// TwinCAT 3 PLC project Demo
// ProgramVersion: 3.1.4023.0
// libraries:
//   Tc2_Standard, * (Beckhoff Automation GmbH)
//   Tc2_System, * (Beckhoff Automation GmbH)
//   Tc3_Module, * (Beckhoff Automation GmbH)
//   VisuSymbols,3.5.10.0,System
// project tree:
//   DUTs/ XeryonDriveError.TcDUT, XeryonDriveSetting.TcDUT, XeryonDriveStatus.TcDUT
//   / GlobalTextList.TcGTLO, PlcTask.TcTTO, Visualization Manager.TcVMO (not stored)
//   GVLs/ GVL.TcGVL
//   POUs/FB/ XeryonDrive.TcPOU
//   POUs/ MAIN.TcPOU, DRIVE_SETTINGS.TcPOU
//   VISUs/ Visualization.TcVIS
// real-time tasks:
//   TASK PlcTask: cycle T#1ms, priority 20, ADS port 350
// I/O:
//   DEVICE Device 1 (EtherCAT), AmsNetId 172.22.11.1.2.1
//     Box 1 (Drive) [Drive]
//     Box 2 (Drive) [Drive] (disabled)
// variable links:
//   Demo/Demo Instance <-> Device 1 (EtherCAT)/Box 1 (Drive)
//     PlcTask Inputs/MAIN.Drive1.iDriveActualPosition <-> Status/Actual position
//     PlcTask Inputs/MAIN.Drive1.iDriveAmplifiersEnabled <-> Status/Amplifiers enabled
//     PlcTask Inputs/MAIN.Drive1.iDriveBusy <-> Status/Execute ack
//     PlcTask Inputs/MAIN.Drive1.iDriveClosedLoop <-> Status/Closed loop
//     PlcTask Inputs/MAIN.Drive1.iDriveEmergencyStop <-> Status/Emergency stop
//     PlcTask Inputs/MAIN.Drive1.iDriveEncoderError <-> Status/Encoder error
//     PlcTask Inputs/MAIN.Drive1.iDriveEncoderIndex <-> Status/Encoder index
//     PlcTask Inputs/MAIN.Drive1.iDriveEncoderValid <-> Status/Encoder valid
//     PlcTask Inputs/MAIN.Drive1.iDriveEndStop <-> Status/End stop
//     PlcTask Inputs/MAIN.Drive1.iDriveErrorCompensation <-> Status/Error compensation
//     PlcTask Inputs/MAIN.Drive1.iDriveErrorLimit <-> Status/Error limit
//     PlcTask Inputs/MAIN.Drive1.iDriveForceZero <-> Status/Force zero
//     PlcTask Inputs/MAIN.Drive1.iDriveLeftEndStop <-> Status/Left end stop
//     PlcTask Inputs/MAIN.Drive1.iDriveMotorOn <-> Status/Motor on
//     PlcTask Inputs/MAIN.Drive1.iDrivePositionFail <-> Status/Position fail
//     PlcTask Inputs/MAIN.Drive1.iDrivePositionReached <-> Status/Position reached
//     PlcTask Inputs/MAIN.Drive1.iDriveRightEndStop <-> Status/Right end stop
//     PlcTask Inputs/MAIN.Drive1.iDriveSafetyTimeoutTriggered <-> Status/Safety timeout
//     PlcTask Inputs/MAIN.Drive1.iDriveScanning <-> Status/Scanning
//     PlcTask Inputs/MAIN.Drive1.iDriveSearchingIndex <-> Status/Searching index
//     PlcTask Inputs/MAIN.Drive1.iDriveSearchingOptimalFrequency <-> Status/Searching optimal frequency
//     PlcTask Inputs/MAIN.Drive1.iDriveSlot <-> Status/Slot
//     PlcTask Inputs/MAIN.Drive1.iDriveThermalProtection1 <-> Status/Thermal protection 1
//     PlcTask Inputs/MAIN.Drive1.iDriveThermalProtection2 <-> Status/Thermal protection 2
//     PlcTask Outputs/MAIN.Drive1.qCommand <-> Position/Command
//     PlcTask Outputs/MAIN.Drive1.qDriveAcc <-> Position/Acceleration
//     PlcTask Outputs/MAIN.Drive1.qDriveDec <-> Position/Deceleration
//     PlcTask Outputs/MAIN.Drive1.qDriveSpeed <-> Position/Speed
//     PlcTask Outputs/MAIN.Drive1.qDriveTargetPos <-> Position/Target position
//     PlcTask Outputs/MAIN.Drive1.qExecute <-> Position/Execute
//   Demo/Demo Instance <-> Device 1 (EtherCAT)/Box 2 (Drive)
//     PlcTask Inputs/MAIN.Drive2.iDriveActualPosition <-> Status/Actual position
//     PlcTask Inputs/MAIN.Drive2.iDriveAmplifiersEnabled <-> Status/Amplifiers enabled
//     PlcTask Inputs/MAIN.Drive2.iDriveBusy <-> Status/Execute ack
//     PlcTask Inputs/MAIN.Drive2.iDriveClosedLoop <-> Status/Closed loop
//     PlcTask Inputs/MAIN.Drive2.iDriveEmergencyStop <-> Status/Emergency stop
//     PlcTask Inputs/MAIN.Drive2.iDriveEncoderError <-> Status/Encoder error
//     PlcTask Inputs/MAIN.Drive2.iDriveEncoderIndex <-> Status/Encoder index
//     PlcTask Inputs/MAIN.Drive2.iDriveEncoderValid <-> Status/Encoder valid
//     PlcTask Inputs/MAIN.Drive2.iDriveEndStop <-> Status/End stop
//     PlcTask Inputs/MAIN.Drive2.iDriveErrorCompensation <-> Status/Error compensation
//     PlcTask Inputs/MAIN.Drive2.iDriveErrorLimit <-> Status/Error limit
//     PlcTask Inputs/MAIN.Drive2.iDriveForceZero <-> Status/Force zero
//     PlcTask Inputs/MAIN.Drive2.iDriveLeftEndStop <-> Status/Left end stop
//     PlcTask Inputs/MAIN.Drive2.iDriveMotorOn <-> Status/Motor on
//     PlcTask Inputs/MAIN.Drive2.iDrivePositionFail <-> Status/Position fail
//     PlcTask Inputs/MAIN.Drive2.iDrivePositionReached <-> Status/Position reached
//     PlcTask Inputs/MAIN.Drive2.iDriveRightEndStop <-> Status/Right end stop
//     PlcTask Inputs/MAIN.Drive2.iDriveSafetyTimeoutTriggered <-> Status/Safety timeout
//     PlcTask Inputs/MAIN.Drive2.iDriveScanning <-> Status/Scanning
//     PlcTask Inputs/MAIN.Drive2.iDriveSearchingIndex <-> Status/Searching index
//     PlcTask Inputs/MAIN.Drive2.iDriveSearchingOptimalFrequency <-> Status/Searching optimal frequency
//     PlcTask Inputs/MAIN.Drive2.iDriveSlot <-> Status/Slot
//     PlcTask Inputs/MAIN.Drive2.iDriveThermalProtection1 <-> Status/Thermal protection 1
//     PlcTask Inputs/MAIN.Drive2.iDriveThermalProtection2 <-> Status/Thermal protection 2
//     PlcTask Outputs/MAIN.Drive2.qCommand <-> Position/Command
//     PlcTask Outputs/MAIN.Drive2.qDriveAcc <-> Position/Acceleration
//     PlcTask Outputs/MAIN.Drive2.qDriveDec <-> Position/Deceleration
//     PlcTask Outputs/MAIN.Drive2.qDriveSpeed <-> Position/Speed
//     PlcTask Outputs/MAIN.Drive2.qDriveTargetPos <-> Position/Target position
//     PlcTask Outputs/MAIN.Drive2.qExecute <-> Position/Execute

CONFIGURATION Demo
    RESOURCE PLC ON TwinCAT3
        TASK PlcTask(INTERVAL := T#1ms, PRIORITY := 20);
        PROGRAM MAIN WITH PlcTask : MAIN;
    END_RESOURCE
END_CONFIGURATION

// ---- DUTs/XeryonDriveError.TcDUT
{attribute 'qualified_only'}
{attribute 'strict'}
{attribute 'to_string'}
TYPE XeryonDriveError :
(
	NO_ERROR := 0,	
	LIMIT_HIT := 1,
	NO_INDEX := 2,
	THERMAL_1 := 3,
	THERMAL_2 := 4,
	ENCODER_ERROR := 5,
	SAFETY_TIMEOUT := 6,
	ERROR_LIMIT := 7,
	ESTOP := 8,
	POS_FAIL := 9,
	DRIVE_DISABLED := 10
);
END_TYPE

// ---- DUTs/XeryonDriveSetting.TcDUT
TYPE XeryonDriveSetting :
STRUCT
	setting : STRING(5);
	value : DINT;
END_STRUCT
END_TYPE

// ---- DUTs/XeryonDriveStatus.TcDUT
{attribute 'qualified_only'}
{attribute 'strict'}
{attribute 'to_string'}
TYPE XeryonDriveStatus :
(	
	Waiting := 0,
	Ready := 1,
	Error := 2,
	SoftError := 3
);
END_TYPE

// ---- GVLs/GVL.TcGVL
{attribute 'qualified_only'}
VAR_GLOBAL	
	Drive1Settings: ARRAY [0..1] OF XeryonDriveSetting;
	Drive2Settings: ARRAY [0..1] OF XeryonDriveSetting;
	Drive3Settings: ARRAY [0..1] OF XeryonDriveSetting;
	Drive4Settings: ARRAY [0..1] OF XeryonDriveSetting;
END_VAR

// ---- POUs/MAIN.TcPOU
PROGRAM MAIN
VAR
	Drive1 : XeryonDrive;
	Drive2 : XeryonDrive;
	Drive3 : XeryonDrive;
	Drive4 : XeryonDrive;
	
	drive1Enable : BOOL;
	drive1EnableOld : BOOL;
	drive1Index : BOOL;
	drive1MoveAbs : BOOL;	
	drive1Dpos : BOOL;		
	drive1Halt : BOOL;
	drive1Stop : BOOL;	
	drive2ResetEncoder : BOOL;	
	drive1ResetEncoder : BOOL;	
	drive1Reset : BOOL;	
	drive1MoveP : BOOL;	
	drive1MoveN : BOOL;		
	drive1JogP : BOOL;	
	drive1JogN : BOOL;	
	drive1Init : BOOL;
	
	drive1State : INT;
	drive1Target : DINT;
	drive1Speed: UDINT := 1000000;
	drive1Acc: UINT := 65535;
	drive1Dec: UINT := 3500;
	drive1ErrorString: STRING;
	
	
	
	drive2Enable : BOOL;
	drive2EnableOld : BOOL;
	drive2Index : BOOL;
	drive2MoveAbs : BOOL;		
	drive2Dpos : BOOL;	
	drive2Halt : BOOL;
	drive2Stop : BOOL;	
	drive2Reset : BOOL;	
	drive2JogP : BOOL;	
	drive2JogN : BOOL;	
	drive2Init : BOOL;
	
	drive2State : INT;
	drive2Target : DINT;
	drive2Speed: UDINT := 150000;
	drive2Acc: UINT := 10000;
	drive2Dec: UINT := 10000;
	
	
	drive3Enable : BOOL;
	drive3EnableOld : BOOL;
	drive3Index : BOOL;
	drive3MoveAbs : BOOL;		
	drive3Dpos : BOOL;		
	drive3Halt : BOOL;
	drive3Stop : BOOL;	
	drive3Reset : BOOL;	
	drive3JogP : BOOL;	
	drive3JogN : BOOL;	
	drive3Init : BOOL;
	
	drive3State : INT;
	drive3Target : DINT;
	drive3Speed: UDINT := 150000;
	drive3Acc: UINT := 10000;
	drive3Dec: UINT := 10000;


	drive4Enable : BOOL;
	drive4EnableOld : BOOL;
	drive4Index : BOOL;
	drive4MoveAbs : BOOL;		
	drive4Dpos : BOOL;		
	drive4Halt : BOOL;
	drive4Stop : BOOL;	
	drive4Reset : BOOL;	
	drive4JogP : BOOL;	
	drive4JogN : BOOL;	
	drive4Init : BOOL;
	
	drive4State : INT;
	drive4Target : DINT;
	drive4Speed: UDINT := 150000;
	drive4Acc: UINT := 10000;
	drive4Dec: UINT := 10000;

	
	target_min : DINT;
	target_max : DINT;
	
	speed_min : DINT;
	speed_max : DINT;
	
	acc_min : DINT;
	acc_max : DINT;
	dec_min : DINT;
	dec_max : DINT;
	
	drive2ErrorString: STRING;
	drive3ErrorString: STRING;
	drive4ErrorString: STRING;
	dpos: DINT;
	drive2MoveN: BOOL;
	Halt: INT;
	drive2MoveP: BOOL;
END_VAR

DRIVE_SETTINGS();

Drive1();
Drive2();
Drive3();
Drive4();
drive1ErrorString := TO_STRING(Drive1.Error);
drive2ErrorString := TO_STRING(Drive2.Error);
drive3ErrorString := TO_STRING(Drive3.Error);
drive4ErrorString := TO_STRING(Drive4.Error);
// DEMO Drive 1
CASE drive1State OF
	0:
		IF(drive1JogP) THEN
			drive1State := 10;
		END_IF
		IF(drive1JogN) THEN
			drive1State := 14;
		END_IF
		IF(drive1MoveP) THEN
			drive1State := 17;
		END_IF
		IF(drive1MoveN) THEN
			drive1State := 20;
		END_IF
		IF(drive1Init) THEN
			drive1State := 9;
		END_IF
		IF(drive1MoveAbs) THEN
			drive1State := 2;
		END_IF
		IF(drive1Index) THEN
			drive1State := 1;
		END_IF
		IF(drive1Dpos) THEN
			drive1State := 8;
		END_IF
	1:
		IF(NOT drive1Index) THEN
			IF(Drive1.Index(drive1Target > 0, drive1Speed, drive1Acc, drive1Dec)<> XeryonDriveStatus.Waiting) THEN
				drive1State := 0;
			END_IF
		END_IF
	2:
		IF(Drive1.MoveAbsolute(dpos, drive1Speed, drive1Acc, drive1Dec)<> XeryonDriveStatus.Waiting) THEN
			IF(dpos < 921600) THEN
				dpos:=dpos+25600;
			ELSE
				dpos := 1000;
			END_IF
			drive1State := 0;
		END_IF
	3:
		IF(Drive1.MoveAbsolute(-40000, drive1Speed, drive1Acc, drive1Dec)<> XeryonDriveStatus.Waiting) THEN
			drive1State := 4;
		END_IF
	4: 
		IF(Drive1.MoveAbsolute(0, drive1Speed, drive1Acc, drive1Dec)<> XeryonDriveStatus.Waiting) THEN
			drive1State := 5;
		END_IF
	5: 
		IF(Drive1.MoveAbsolute(-10000, drive1Speed, drive1Acc, drive1Dec)<> XeryonDriveStatus.Waiting) THEN
			drive1State := 6;
		END_IF
	6: 
		IF(Drive1.MoveAbsolute(0, drive1Speed, drive1Acc, drive1Dec)<> XeryonDriveStatus.Waiting) THEN
			drive1State := 7;
		END_IF		
	7: 
		IF(Drive1.MoveAbsolute(-5000, drive1Speed, drive1Acc, drive1Dec)<> XeryonDriveStatus.Waiting) THEN
			drive1State := 0;
		END_IF
	8:
		IF(NOT drive1Dpos) THEN
			IF(Drive1.MoveAbsolute(drive1Target, drive1Speed, drive1Acc, drive1Dec)<> XeryonDriveStatus.Waiting) THEN
				drive1State := 0;
			END_IF
		END_IF
	9:
		IF(Drive1.Init(GVL.Drive1Settings) = TRUE) THEN
			drive1State := 0;
		END_IF
	10:
		IF(Drive1.Scan(TRUE, drive1Speed, drive1Acc, drive1Dec) <>  XeryonDriveStatus.Waiting) THEN
			drive1State := 12;
		END_IF
	12: //TBD GST : why is this state needed???
		IF(NOT drive1JogP) THEN
			drive1State := 13;
		END_IF
	13:
		IF(Drive1.Halt() <>  XeryonDriveStatus.Waiting) THEN
			drive1State := 0;
		END_IF
	14:
		IF(Drive1.Scan(FALSE, drive1Speed, drive1Acc, drive1Dec) <>  XeryonDriveStatus.Waiting) THEN
			drive1State := 15;
		END_IF
	15:
		IF(NOT drive1JogN) THEN
			drive1State := 16;
		END_IF
	16:
		IF(Drive1.Halt() <>  XeryonDriveStatus.Waiting) THEN
			drive1State := 0;
		END_IF
		
	17:
		IF(Drive1.MoveOpen(TRUE) <>  XeryonDriveStatus.Waiting) THEN
			drive1State := 18;
		END_IF
	18:
		IF(NOT drive1MoveP) THEN
			drive1State := 19;
		END_IF
	19:
		IF(Drive1.Halt() <>  XeryonDriveStatus.Waiting) THEN
			drive1State := 0;
		END_IF
	20:
		IF(Drive1.MoveOpen(FALSE) <>  XeryonDriveStatus.Waiting) THEN
			drive1State := 21;
		END_IF
	21:
		IF(NOT drive1MoveN) THEN
			drive1State := 22;
		END_IF
	22:
		IF(Drive1.Halt() <>  XeryonDriveStatus.Waiting) THEN
			drive1State := 0;
		END_IF	
			
END_CASE

IF(drive1Halt) THEN
	Drive1.Halt();
END_IF
IF(drive1Enable <> drive1EnableOld) THEN	
	IF(Drive1.Enable(drive1Enable) <> XeryonDriveStatus.Waiting) THEN
		drive1EnableOld := drive1Enable;	
	END_IF
END_IF
IF(drive1Stop) THEN
	Drive1.Stop();
END_IF
IF(drive1Reset) THEN
	Drive1.Reset();
END_IF
IF(drive1ResetEncoder) THEN
	Drive1.ResetEncoder();
END_IF

// DEMO Drive 2
CASE drive2State OF
	0:
		IF(drive2JogP) THEN
			drive2State := 10;
		END_IF
		IF(drive2JogN) THEN
			drive2State := 14;
		END_IF
		IF(drive2MoveP) THEN
			drive2State := 17;
		END_IF
		IF(drive2MoveN) THEN
			drive2State := 20;
		END_IF
		IF(drive2Init) THEN
			drive2State := 9;
		END_IF
		IF(drive2MoveAbs) THEN
			drive2State := 2;
		END_IF
		IF(drive2Index) THEN
			drive2State := 1;
		END_IF
		IF(drive2Dpos) THEN
			drive2State := 8;
		END_IF
	1:
		IF(NOT drive2Index) THEN
			IF(Drive2.Index(drive2Target > 0, drive2Speed, drive2Acc, drive2Dec)<> XeryonDriveStatus.Waiting) THEN
				drive2State := 0;
			END_IF
		END_IF
	2:
		IF(Drive2.MoveAbsolute(40000, drive2Speed, drive2Acc, drive2Dec)<> XeryonDriveStatus.Waiting) THEN
			drive2State := 3;
		END_IF
	3: 
		IF(Drive2.MoveAbsolute(0, drive2Speed, drive2Acc, drive2Dec)<> XeryonDriveStatus.Waiting) THEN
			drive2State := 4;
		END_IF
	4: 
		IF(Drive2.MoveAbsolute(-40000, drive2Speed, drive2Acc, drive2Dec)<> XeryonDriveStatus.Waiting) THEN
			drive2State := 5;
		END_IF
	5: 
		IF(Drive2.MoveAbsolute(-10000, drive2Speed, drive2Acc, drive2Dec)<> XeryonDriveStatus.Waiting) THEN
			drive2State := 6;
		END_IF
	6: 
		IF(Drive2.MoveAbsolute(-5000, drive2Speed, drive2Acc, drive2Dec)<> XeryonDriveStatus.Waiting) THEN
			drive2State := 7;
		END_IF		
	7: 
		IF(Drive2.MoveAbsolute(0, drive2Speed, drive2Acc, drive2Dec)<> XeryonDriveStatus.Waiting) THEN
			drive2State := 0;
		END_IF
	8:
		IF(NOT drive2Dpos) THEN
			IF(Drive2.MoveAbsolute(drive2Target, drive2Speed, drive2Acc, drive2Dec)<> XeryonDriveStatus.Waiting) THEN
				drive2State := 0;
			END_IF
		END_IF
	9:
		IF(Drive2.Init(GVL.Drive2Settings) = TRUE) THEN
			drive2State := 0;
		END_IF
	10:
		IF(Drive2.Scan(TRUE, drive2Speed, drive2Acc, drive2Dec) <>  XeryonDriveStatus.Waiting) THEN
			drive2State := 12;
		END_IF
	12:
		IF(NOT drive2JogP) THEN
			drive2State := 13;
		END_IF
	13:
		IF(Drive2.Halt() <>  XeryonDriveStatus.Waiting) THEN
			drive2State := 0;
		END_IF
	14:
		IF(Drive2.Scan(FALSE, drive2Speed, drive2Acc, drive2Dec) <>  XeryonDriveStatus.Waiting) THEN
			drive2State := 15;
		END_IF
	15:
		IF(NOT drive2JogN) THEN
			drive2State := 16;
		END_IF
	16:
		IF(Drive2.Halt() <>  XeryonDriveStatus.Waiting) THEN
			drive2State := 0;
		END_IF
	17:
		IF(Drive2.MoveOpen(TRUE) <>  XeryonDriveStatus.Waiting) THEN
			drive2State := 18;
		END_IF
	18:
		IF(NOT drive2MoveP) THEN
			drive2State := 19;
		END_IF
	19:
		IF(Drive2.Halt() <>  XeryonDriveStatus.Waiting) THEN
			drive2State := 0;
		END_IF
	20:
		IF(Drive2.MoveOpen(FALSE) <>  XeryonDriveStatus.Waiting) THEN
			drive2State := 21;
		END_IF
	21:
		IF(NOT drive2MoveN) THEN
			drive2State := 22;
		END_IF
	22:
		IF(Drive2.Halt() <>  XeryonDriveStatus.Waiting) THEN
			drive2State := 0;
		END_IF
END_CASE

IF(drive2Halt) THEN
	Drive2.Halt();
END_IF
IF(drive2Enable <> drive2EnableOld) THEN
	IF(Drive2.Enable(drive2Enable) <> XeryonDriveStatus.Waiting) THEN
		drive2EnableOld := drive2Enable;	
	END_IF
END_IF
IF(drive2Stop) THEN
	Drive2.Stop();
END_IF
IF(drive2Reset) THEN
	Drive2.Reset();
END_IF
IF(drive2ResetEncoder) THEN
	Drive2.ResetEncoder();
END_IF

// DEMO Drive 3
CASE drive3State OF
	0:
		IF(drive3JogP) THEN
			drive3State := 10;
		END_IF
		IF(drive3JogN) THEN
			drive3State := 14;
		END_IF
		IF(drive3Init) THEN
			drive3State := 9;
		END_IF
		IF(drive3MoveAbs) THEN
			drive3State := 2;
		END_IF
		IF(drive3Index) THEN
			drive3State := 1;
		END_IF
		IF(drive3Dpos) THEN
			drive3State := 8;
		END_IF
	1:
		IF(NOT drive3Index) THEN
			IF(Drive3.Index(drive3Target  > 0, drive3Speed, drive3Acc, drive3Dec) <> XeryonDriveStatus.Waiting) THEN
				drive3State := 0;
			END_IF
		END_IF
	2:
		IF(Drive3.MoveAbsolute(40000, drive3Speed, drive3Acc, drive3Dec) <> XeryonDriveStatus.Waiting) THEN
			drive3State := 3;
		END_IF
	3: 
		IF(Drive3.MoveAbsolute(0, drive3Speed, drive3Acc, drive3Dec) <> XeryonDriveStatus.Waiting) THEN
			drive3State := 4;
		END_IF
	4: 
		IF(Drive3.MoveAbsolute(-40000, drive3Speed, drive3Acc, drive3Dec) <> XeryonDriveStatus.Waiting) THEN
			drive3State := 5;
		END_IF
	5: 
		IF(Drive3.MoveAbsolute(15000, drive3Speed, drive3Acc, drive3Dec) <> XeryonDriveStatus.Waiting) THEN
			drive3State := 6;
		END_IF
	6: 
		IF(Drive3.MoveAbsolute(-15000, drive3Speed, drive3Acc, drive3Dec) <> XeryonDriveStatus.Waiting) THEN
			drive3State := 7;
		END_IF		
	7: 
		IF(Drive3.MoveAbsolute(0, drive3Speed, drive3Acc, drive3Dec) <> XeryonDriveStatus.Waiting) THEN
			drive3State := 0;
		END_IF
	8:
		IF(NOT drive3Dpos) THEN
			IF(Drive3.MoveAbsolute(drive3Target, drive3Speed, drive3Acc, drive3Dec) <> XeryonDriveStatus.Waiting) THEN
				drive3State := 0;
			END_IF
		END_IF
	9:
		IF(Drive3.Init(GVL.Drive3Settings) = TRUE) THEN
			drive3State := 0;
		END_IF
	10:
		IF(Drive3.Scan(TRUE, drive3Speed, drive3Acc, drive3Dec) <>  XeryonDriveStatus.Waiting) THEN
			drive3State := 12;
		END_IF
	12:
		IF(NOT drive3JogP) THEN
			drive3State := 13;
		END_IF
	13:
		IF(Drive3.Halt() <>  XeryonDriveStatus.Waiting) THEN
			drive3State := 0;
		END_IF
	14:
		IF(Drive3.Scan(FALSE, drive3Speed, drive3Acc, drive3Dec) <>  XeryonDriveStatus.Waiting) THEN
			drive3State := 15;
		END_IF
	15:
		IF(NOT drive3JogN) THEN
			drive3State := 16;
		END_IF
	16:
		IF(Drive3.Halt() <>  XeryonDriveStatus.Waiting) THEN
			drive3State := 0;
		END_IF		
		
END_CASE

IF(drive3Halt) THEN
	Drive3.Halt();
END_IF
IF(drive3Stop) THEN
	Drive3.Stop();
END_IF
IF(drive3Enable <> drive3EnableOld) THEN
	IF(Drive3.Enable(drive3Enable) <> XeryonDriveStatus.Waiting) THEN
		drive3EnableOld := drive3Enable;	
	END_IF
END_IF
IF(drive3Reset) THEN
	Drive3.Reset();
END_IF




// DEMO Drive 4
CASE drive4State OF
	0:
		IF(drive4JogP) THEN
			drive4State := 10;
		END_IF
		IF(drive4JogN) THEN
			drive4State := 14;
		END_IF
		IF(drive4Init) THEN
			drive4State := 9;
		END_IF
		IF(drive4MoveAbs) THEN
			drive4State := 2;
		END_IF
		IF(drive4Index) THEN
			drive4State := 1;
		END_IF
		IF(drive4Dpos) THEN
			drive4State := 8;
		END_IF
	1:
		IF(NOT drive4Index) THEN
			IF(Drive4.Index(drive4Target  > 0, drive4Speed, drive4Acc, drive4Dec) <> XeryonDriveStatus.Waiting) THEN
				drive4State := 0;
			END_IF
		END_IF
	2:
		IF(Drive4.MoveAbsolute(0, drive4Speed, drive4Acc, drive4Dec) <> XeryonDriveStatus.Waiting) THEN
			drive4State := 3;
		END_IF
	3: 
		IF(Drive4.MoveAbsolute(35000, drive4Speed, drive4Acc, drive4Dec) <> XeryonDriveStatus.Waiting) THEN
			drive4State := 4;
		END_IF
	4: 
		IF(Drive4.MoveAbsolute(0, drive4Speed, drive4Acc, drive4Dec) <> XeryonDriveStatus.Waiting) THEN
			drive4State := 5;
		END_IF
	5: 
		IF(Drive4.MoveAbsolute(-35000, drive4Speed, drive4Acc, drive4Dec) <> XeryonDriveStatus.Waiting) THEN
			drive4State := 6;
		END_IF
	6: 
		IF(Drive4.MoveAbsolute(0, drive4Speed, drive4Acc, drive4Dec) <> XeryonDriveStatus.Waiting) THEN
			drive4State := 7;
		END_IF		
	7: 
		IF(Drive4.MoveAbsolute(35000, drive4Speed, drive4Acc, drive4Dec) <> XeryonDriveStatus.Waiting) THEN
			drive4State := 0;
		END_IF
	8:
		IF(NOT drive4Dpos) THEN
			IF(Drive4.MoveAbsolute(drive4Target, drive4Speed, drive4Acc, drive4Dec) <> XeryonDriveStatus.Waiting) THEN
				drive4State := 0;
			END_IF
		END_IF
	9:
		IF(Drive4.Init(GVL.Drive4Settings) = TRUE) THEN
			drive4State := 0;
		END_IF
	10:
		IF(Drive4.Scan(TRUE, drive4Speed, drive4Acc, drive4Dec) <>  XeryonDriveStatus.Waiting) THEN
			drive4State := 12;
		END_IF
	12:
		IF(NOT drive4JogP) THEN
			drive4State := 13;
		END_IF
	13:
		IF(Drive4.Halt() <>  XeryonDriveStatus.Waiting) THEN
			drive4State := 0;
		END_IF
	14:
		IF(Drive4.Scan(FALSE, drive4Speed, drive4Acc, drive4Dec) <>  XeryonDriveStatus.Waiting) THEN
			drive4State := 15;
		END_IF
	15:
		IF(NOT drive4JogN) THEN
			drive4State := 16;
		END_IF
	16:
		IF(Drive4.Halt() <>  XeryonDriveStatus.Waiting) THEN
			drive4State := 0;
		END_IF		
		
END_CASE

IF(drive4Halt) THEN
	Drive4.Halt();
END_IF
IF(drive4Stop) THEN
	Drive4.Stop();
END_IF
IF(drive4Enable <> drive4EnableOld) THEN
	IF(Drive4.Enable(drive4Enable) <> XeryonDriveStatus.Waiting) THEN
		drive4EnableOld := drive4Enable;	
	END_IF
END_IF
IF(drive4Reset) THEN
	Drive4.Reset();
END_IF


target_max := 1843200;
target_min := -1843200;

speed_min := 0;
speed_max := 1000000;


acc_min := 0;
acc_max := 65535;

dec_min := 0;
dec_max := 65535;

END_PROGRAM

// ---- POUs/FB/XeryonDrive.TcPOU
FUNCTION_BLOCK XeryonDrive
VAR_INPUT
END_VAR
VAR_OUTPUT
	ActPosition : DINT;
	Done : BOOL;
	Busy : BOOL;
	HasError : BOOL;
	HasIndex : BOOL;
	Error : XeryonDriveError;
	MotorOn : BOOL;
	LeftEndstop : BOOL;
	RightEndstop : BOOL;
END_VAR
VAR
	iDriveActualPosition AT %I* : DINT;
	iDriveAmplifiersEnabled AT %I* : BOOL;
	iDriveEndStop AT %I* : BOOL;
	iDriveThermalProtection1 AT %I* : BOOL;
	iDriveThermalProtection2 AT %I* : BOOL;
	iDriveForceZero AT %I* : BOOL;
	iDriveMotorOn AT %I* : BOOL;
	iDriveClosedLoop AT %I* : BOOL;
	iDriveEncoderIndex AT %I* : BOOL;
	iDriveEncoderValid AT %I* : BOOL;
	iDriveSearchingIndex AT %I* : BOOL;
	iDrivePositionReached AT %I* : BOOL;
	iDriveErrorCompensation AT %I* : BOOL;
	iDriveEncoderError AT %I* : BOOL;
	iDriveScanning AT %I* : BOOL;
	iDriveLeftEndStop AT %I* : BOOL;
	iDriveRightEndStop AT %I* : BOOL;
	iDriveErrorLimit AT %I* : BOOL;
	iDriveSearchingOptimalFrequency AT %I* : BOOL;
	iDriveSafetyTimeoutTriggered AT %I* : BOOL;
	iDriveBusy AT %I* : BOOL;
	iDriveEmergencyStop AT %I* : BOOL;
	iDrivePositionFail AT %I* : BOOL;
	iDriveSlot AT %I* : USINT;
	
	qDriveTargetPos AT %Q* : DINT;
	qDriveSpeed AT %Q* : DINT;
	qDriveAcc AT %Q* : INT;
	qDriveDec AT %Q* : INT;
	qCommand AT %Q* : STRING(4);
	qExecute AT %Q* : USINT;
	
	
	new_TargetPos : DINT;
	new_Speed : UDINT;
	new_Acc : INT;
	new_Dec : INT;
	new_command : STRING(4);
	
	state : INT := 0;
	command_start : BOOL;
	command_done : BOOL;
	command_irq : BOOL;
	init_state : INT := -1;
	
	has_index : BOOL;
	
END_VAR

has_index := iDriveEncoderValid;
ActPosition := iDriveActualPosition;
MotorOn := iDriveMotorOn;
LeftEndstop := iDriveLeftEndStop;
RightEndstop := iDriveRightEndStop;
HasIndex := has_index;

// Check error bits
IF(iDriveThermalProtection1) THEN
	HasError := TRUE;
	Error := XeryonDriveError.THERMAL_1;
END_IF
IF(iDriveThermalProtection1) THEN
	HasError := TRUE;
	Error := XeryonDriveError.THERMAL_2;
END_IF
IF(iDriveEncoderError) THEN
	HasError := TRUE;
	Error := XeryonDriveError.ENCODER_ERROR;
END_IF
IF(iDriveEmergencyStop) THEN
	HasError := TRUE;
	Error := XeryonDriveError.ESTOP;
END_IF
IF(iDriveErrorLimit) THEN
	HasError := TRUE;
	Error := XeryonDriveError.ERROR_LIMIT;
END_IF

CASE state OF
	0: // Idle
	 	IF(command_irq = TRUE) THEN
			state := 4;
		END_IF
	 	IF(command_start = TRUE) THEN
			state := 1;
		END_IF
		Busy := FALSE;
	1:
		Busy := TRUE;
		Done := FALSE;
		qCommand := new_command;
		qDriveTargetPos := new_TargetPos;
		qDriveSpeed := UDINT_TO_DINT(new_Speed);
		qDriveAcc := new_Acc;
		qDriveDec := new_Dec;
		qExecute := 255;
		command_start := FALSE;
		command_done := FALSE;
		IF(iDriveBusy = TRUE) THEN
			qExecute := 0;
			state := 2;	
		END_IF		
	2:	
		IF(iDriveBusy = FALSE) THEN
			state := 3;	
		END_IF	
	3: 	IF(command_done = TRUE) THEN
			state := 0;			
			Done := TRUE;
		END_IF
	 	IF(command_irq = TRUE) THEN
			state := 4;
		END_IF
	// Interrupt commands 
	4:	
		command_irq := FALSE;
		Busy := TRUE;
		Done := FALSE;
		qCommand := new_command;
		qDriveTargetPos := new_TargetPos;
		qDriveSpeed := UDINT_TO_DINT(new_Speed);
		qDriveAcc := new_Acc;
		qDriveDec := new_Dec;
		qExecute := 255;
		command_start := FALSE;
		command_done := FALSE;
		IF(iDriveBusy = TRUE) THEN
			qExecute := 0;
			state := 5;	
		END_IF		
	5:	IF(iDriveBusy = FALSE) THEN
			qExecute := 0;
			state := 6;	
		END_IF	
	6:
		state := 0;			
		Done := TRUE;
	
END_CASE

METHOD CheckError : BOOL
VAR_INPUT
END_VAR
CheckError := FALSE;
// Only check these two  bits when moving
IF(iDrivePositionFail) THEN
	HasError := TRUE;
	Error := XeryonDriveError.POS_FAIL;
END_IF
IF(iDriveSafetyTimeoutTriggered) THEN
	HasError := TRUE;
	Error := XeryonDriveError.SAFETY_TIMEOUT;
END_IF
IF(HasError) THEN
	CheckError := TRUE;	
END_IF
END_METHOD

ACTION ClearError:
HasError := FALSE;
Error := XeryonDriveError.NO_ERROR;

// Reset the index when clearing the error
IF(iDriveEncoderValid) THEN
	has_index := TRUE;
ELSE
	has_index := FALSE;
END_IF
END_ACTION

METHOD Enable : XeryonDriveStatus
VAR_INPUT
	val : BOOL;
END_VAR
Enable := XeryonDriveStatus.Waiting;
IF(state = 0) OR (state = 3) THEN
	new_command := 'ENBL';
	IF(val) THEN
		new_TargetPos := 1;
	ELSE
		new_TargetPos := 0;
	END_IF
	command_start := TRUE;
	command_irq := TRUE;
END_IF
IF(state = 6) THEN
	command_done := TRUE;
	Enable := XeryonDriveStatus.Ready;
	// Clear error
	IF(val) THEN
		ClearError();
	END_IF	
END_IF
END_METHOD

METHOD Halt : XeryonDriveStatus
VAR_INPUT
END_VAR
Halt := XeryonDriveStatus.Waiting;
IF(state = 0) OR (state = 3)THEN
	new_command := 'HALT';
	command_start := TRUE;
	command_irq := TRUE;
END_IF
IF(state = 6) THEN
	command_done := TRUE;
	Halt := XeryonDriveStatus.Ready;
END_IF
END_METHOD

METHOD Index : XeryonDriveStatus
VAR_INPUT
	Direction : BOOL;
	Velocity : UDINT;
	Acceleration: UINT;
	Deceleration: UINT;
END_VAR
Index := XeryonDriveStatus.Waiting;
IF(state = 0) THEN
	// Only execute when we don't have an active error
	IF(NOT HasError) THEN
		IF(iDriveAmplifiersEnabled) THEN
			new_command := 'INDX';
			IF(Direction) THEN
				new_TargetPos := +1;	
			ELSE
				new_TargetPos := -1;
			END_IF		
			new_Speed := Velocity;
			new_Acc := UINT_TO_INT(Acceleration);
			new_Dec := UINT_TO_INT(Deceleration);
			command_start := TRUE;
		ELSE
			
			HasError := TRUE;
			IF(NOT iDriveAmplifiersEnabled) THEN
				Error := XeryonDriveError.DRIVE_DISABLED;	
			END_IF		
			Index := XeryonDriveStatus.Error;	
		END_IF
	ELSE
		Index := XeryonDriveStatus.Error;
	END_IF
END_IF
IF(state = 3) THEN
	// Normal flow, when index is found --> ready 
	IF(iDriveEncoderValid) THEN
		command_done := TRUE;
		Index := XeryonDriveStatus.Ready;
	END_IF
	
	// When hitting the endstop signal a SoftError, doesn't need a reset, but limit the motion
	IF(iDriveEndstop) THEN
		command_done := TRUE;
		Index := XeryonDriveStatus.SoftError;		
	END_IF
	
	// Handle drive errors
	IF(CheckError()) THEN
		command_done := TRUE;
		Index := XeryonDriveStatus.Error;
	END_IF
END_IF
IF(state = 6) THEN
	Index := XeryonDriveStatus.Ready;
END_IF
END_METHOD

METHOD Init : BOOL
VAR_IN_OUT
	settings : ARRAY[*] OF XeryonDriveSetting;
END_VAR
Init := FALSE;

// Start
IF(init_state = -1) THEN
	init_state := DINT_TO_INT(LOWER_BOUND(settings, 1));
END_IF

IF(init_state >=  LOWER_BOUND(settings, 1)) AND (init_state < UPPER_BOUND(settings, 1))  THEN
	IF(Write(settings[init_state].setting, settings[init_state].value) <> XeryonDriveStatus.Waiting) THEN
		init_state := init_state + 1;
		IF(init_state = UPPER_BOUND(settings, 1)) THEN
			init_state := -1;
			Init := TRUE;
		END_IF
	END_IF
END_IF
END_METHOD

METHOD MoveAbsolute : XeryonDriveStatus
VAR_INPUT
	Position : DINT;
	Velocity : UDINT;
	Acceleration: UINT;
	Deceleration: UINT;
	
END_VAR
MoveAbsolute := XeryonDriveStatus.Waiting;
IF(state = 0) THEN
	// Only execute when we don't have an active error
	IF(NOT HasError) THEN		
		// Check if we have an index
		IF(has_index) AND iDriveAmplifiersEnabled THEN
			new_command := 'DPOS';
			new_TargetPos := Position;
			new_Speed := Velocity;
			new_Acc := UINT_TO_INT(Acceleration);
			new_Dec := UINT_TO_INT(Deceleration);
			command_start := TRUE;
		ELSE
			HasError := TRUE;
			IF(NOT has_index) THEN
				Error := XeryonDriveError.NO_INDEX;	
			END_IF
			IF(NOT iDriveAmplifiersEnabled) THEN
				Error := XeryonDriveError.DRIVE_DISABLED;	
			END_IF

			MoveAbsolute := XeryonDriveStatus.Error;
		END_IF
	ELSE
		MoveAbsolute := XeryonDriveStatus.Error;
	END_IF	
	
END_IF
IF(state = 3) THEN
	
	// Normal flow, when position is reached  --> ready 
	IF(iDrivePositionReached) THEN
		command_done := TRUE;
		MoveAbsolute := XeryonDriveStatus.Ready;
	END_IF
	
	// When hitting the endstop signal a SoftError, doesn't need a reset, but limit the motion
	IF(iDriveEndstop) THEN
		command_done := TRUE;
		MoveAbsolute := XeryonDriveStatus.SoftError;		
	END_IF
	
	// Handle drive errors
	IF(CheckError()) THEN
		command_done := TRUE;
		MoveAbsolute := XeryonDriveStatus.Error;
	END_IF
	
END_IF
IF(state = 6) THEN
	MoveAbsolute := XeryonDriveStatus.Ready;
END_IF
END_METHOD

METHOD MoveOpen : XeryonDriveStatus
VAR_INPUT
	Direction: BOOL;	
END_VAR
MoveOpen := XeryonDriveStatus.Waiting;
IF(state = 0) THEN
	IF( NOT HasError) THEN
		IF iDriveAmplifiersEnabled THEN
			new_command := 'MOVE';
			IF(Direction) THEN
				new_TargetPos := +1;	
			ELSE
				new_TargetPos := -1;
			END_IF
			new_Speed := 0;
			new_Acc := UINT_TO_INT(0);
			new_Dec := UINT_TO_INT(0);
			command_start := TRUE;
		ELSE
			HasError := TRUE;
			IF(NOT iDriveAmplifiersEnabled) THEN
				Error := XeryonDriveError.DRIVE_DISABLED;	
			END_IF		
			MoveOpen := XeryonDriveStatus.Error;	
		END_IF
	ELSE
		MoveOpen := XeryonDriveStatus.Error;
	END_IF	
END_IF
IF(state = 3) THEN
	command_done := TRUE;
	MoveOpen := XeryonDriveStatus.Ready;
END_IF
IF(state = 6) THEN
	MoveOpen := XeryonDriveStatus.Ready;
END_IF
END_METHOD

METHOD Reset : XeryonDriveStatus
VAR_INPUT
END_VAR
Reset := XeryonDriveStatus.Waiting;
IF(state = 0) OR (state = 3) THEN
	new_command := 'RSET';
	command_start := TRUE;
	command_irq := TRUE;
END_IF
IF(state = 6) THEN
	command_done := TRUE;
	Reset := XeryonDriveStatus.Ready;
	
	// Clear errors
	ClearError();
	
	// Clear Index
	has_index := FALSE;
	
END_IF
END_METHOD

METHOD ResetEncoder : XeryonDriveStatus
ResetEncoder := XeryonDriveStatus.Waiting;
IF(state = 0) OR (state = 3) THEN
	new_command := 'ENCR';
	command_start := TRUE;
	command_irq := TRUE;
END_IF
IF(state = 6) THEN
	command_done := TRUE;
	ResetEncoder := XeryonDriveStatus.Ready;
	
	// Clear Index
	has_index := FALSE;
	
END_IF
END_METHOD

METHOD Scan : XeryonDriveStatus
VAR_INPUT
	Direction: BOOL;
	Velocity : UDINT;
	Acceleration: UINT;
	Deceleration: UINT;
END_VAR
Scan := XeryonDriveStatus.Waiting;
IF(state = 0) THEN
	IF( NOT HasError) THEN
		IF iDriveAmplifiersEnabled THEN
			new_command := 'SCAN';
			IF(Direction) THEN
				new_TargetPos := +1;	
			ELSE
				new_TargetPos := -1;
			END_IF
			new_Speed := Velocity;
			new_Acc := UINT_TO_INT(Acceleration);
			new_Dec := UINT_TO_INT(Deceleration);
			command_start := TRUE;
		ELSE
			HasError := TRUE;
			IF(NOT iDriveAmplifiersEnabled) THEN
				Error := XeryonDriveError.DRIVE_DISABLED;	
			END_IF		
			Scan := XeryonDriveStatus.Error;	
		END_IF
	ELSE
		Scan := XeryonDriveStatus.Error;
	END_IF	
END_IF
IF(state = 3) THEN
	// Normal flow, when end stop is reached  --> ready 
	IF(((new_TargetPos = +1) AND (iDriveRightEndStop)) OR 
	   ((new_TargetPos = -1) AND (iDriveLeftEndStop))) THEN
		command_done := TRUE;
		Scan := XeryonDriveStatus.Ready;
	END_IF
	
	// Handle drive errors
	IF(CheckError()) THEN
		command_done := TRUE;
		Scan := XeryonDriveStatus.Error;
	END_IF	
END_IF
IF(state = 6) THEN
	Scan := XeryonDriveStatus.Ready;
END_IF
END_METHOD

METHOD Stop : XeryonDriveStatus
VAR_INPUT
END_VAR
Stop := XeryonDriveStatus.Waiting;
IF(state = 0) OR (state = 3) THEN
	new_command := 'STOP';
	command_start := TRUE;
	command_irq := TRUE;
END_IF
IF(state = 6) THEN
	command_done := TRUE;
	Stop := XeryonDriveStatus.Ready;
	
END_IF
END_METHOD

METHOD Write : XeryonDriveStatus
VAR_INPUT
	setting : STRING(4);
	value : DINT;
END_VAR
Write := XeryonDriveStatus.Waiting;
IF(state = 0) THEN
	new_command := setting;
	new_TargetPos := value;
	new_Speed := 0;
	new_Acc := 0;
	new_Dec := 0;
	command_start := TRUE;
END_IF
IF(state = 3) THEN
	command_done := TRUE;
	Write := XeryonDriveStatus.Ready;
END_IF
END_METHOD

END_FUNCTION_BLOCK

// ---- POUs/DRIVE_SETTINGS.TcPOU
PROGRAM DRIVE_SETTINGS
VAR
	init : BOOL := FALSE;
	delta_zone: DINT;
END_VAR

IF init = FALSE THEN
init := TRUE;

// Drive 1
GVL.Drive1Settings[0].setting:='4PHS';
GVL.Drive1Settings[0].value:=0;
//GVL.Drive1Settings[1].setting:='LLIM';
//GVL.Drive1Settings[1].value:=-2000000;
//GVL.Drive1Settings[2].setting:='HLIM';
//GVL.Drive1Settings[2].value:=2000000;
//GVL.Drive1Settings[3].setting:='ENCD';
//GVL.Drive1Settings[3].value:=1;
//GVL.Drive1Settings[4].setting:='ENCO';
//GVL.Drive1Settings[4].value:=0;
//GVL.Drive1Settings[5].setting:='INDA';
//GVL.Drive1Settings[5].value:=1;
//GVL.Drive1Settings[6].setting:='ISPD';
//GVL.Drive1Settings[6].value:=5000;
//GVL.Drive1Settings[7].setting:='ILIM';
//GVL.Drive1Settings[7].value:=30000;
//GVL.Drive1Settings[8].setting:='FILE';
//GVL.Drive1Settings[8].value:=0;
//GVL.Drive1Settings[9].setting:='ZON1';
//GVL.Drive1Settings[9].value:=1000;
//GVL.Drive1Settings[10].setting:='ZON2';
//GVL.Drive1Settings[10].value:=10000;
//delta_zone := GVL.Drive1Settings[10].value - GVL.Drive1Settings[9].value;
//GVL.Drive1Settings[11].setting:='FREQ';
//GVL.Drive1Settings[11].value:=173000;
//GVL.Drive1Settings[12].setting:='FRQ2';
//GVL.Drive1Settings[12].value:=172000;
//GVL.Drive1Settings[13].setting:='FRAT';
//IF delta_zone = 0 THEN
//	GVL.Drive1Settings[13].value:=0;
//ELSE
//	GVL.Drive1Settings[13].value:= 65536 * (GVL.Drive1Settings[11].value - GVL.Drive1Settings[12].value) / delta_zone;	//145635;
//END_IF
//GVL.Drive1Settings[14].setting:='PROP';
//GVL.Drive1Settings[14].value:=120;
//GVL.Drive1Settings[15].setting:='PRO2';
//GVL.Drive1Settings[15].value:=90;
//GVL.Drive1Settings[16].setting:='PRAT';
//IF delta_zone = 0 THEN
//	GVL.Drive1Settings[16].value:=0;
//ELSE
//	GVL.Drive1Settings[16].value:= 65536 * (GVL.Drive1Settings[14].value - GVL.Drive1Settings[15].value) / delta_zone;	//2184;
//END_IF
//GVL.Drive1Settings[17].setting:='INTF';
//GVL.Drive1Settings[17].value:=15; //15
//GVL.Drive1Settings[18].setting:='CFRQ';
//GVL.Drive1Settings[18].value:=60000; //100000
//GVL.Drive1Settings[19].setting:='DUCO';
//GVL.Drive1Settings[19].value:=0; //1
//GVL.Drive1Settings[20].setting:='PTOL';
//GVL.Drive1Settings[20].value:=100;
//GVL.Drive1Settings[21].setting:='PTO2';
//GVL.Drive1Settings[21].value:=160;
//GVL.Drive1Settings[22].setting:='PHAC';
//GVL.Drive1Settings[22].value:=0;
//GVL.Drive1Settings[23].setting:='MIMP';
//GVL.Drive1Settings[23].value:=5000; //5000
//GVL.Drive1Settings[24].setting:='MAMP';
//GVL.Drive1Settings[24].value:=65535;
//GVL.Drive1Settings[25].setting:='SLOP';
//GVL.Drive1Settings[25].value:= (GVL.Drive1Settings[24].value - GVL.Drive1Settings[23].value) / 192; //312;
//GVL.Drive1Settings[26].setting:='SOFS';
//GVL.Drive1Settings[26].value:= GVL.Drive1Settings[23].value - 64 * GVL.Drive1Settings[25].value; //-14968;
//GVL.Drive1Settings[27].setting:='FILA';
//GVL.Drive1Settings[27].value:=1; //1
//GVL.Drive1Settings[28].setting:='FILP';
//GVL.Drive1Settings[28].value:=1; //1
//GVL.Drive1Settings[29].setting:='AMPL';
//GVL.Drive1Settings[29].value:=65535;
//GVL.Drive1Settings[30].setting:='PHAS';
//GVL.Drive1Settings[30].value:=16383;
//GVL.Drive1Settings[31].setting:='TOUT';
//GVL.Drive1Settings[31].value:=500;
//GVL.Drive1Settings[32].setting:='TOU2';
//GVL.Drive1Settings[32].value:=0;
//GVL.Drive1Settings[33].setting:='TOU3';
//GVL.Drive1Settings[33].value:=7000;
//GVL.Drive1Settings[34].setting:='ELIM';
//GVL.Drive1Settings[34].value:=0;
//GVL.Drive1Settings[35].setting:='BLCK';
//GVL.Drive1Settings[35].value:=0;
//GVL.Drive1Settings[36].setting:='DLAY';
//GVL.Drive1Settings[36].value:=0;
//GVL.Drive1Settings[37].setting:='DTIM';
//GVL.Drive1Settings[37].value:=0;
//GVL.Drive1Settings[38].setting:='SSPD';
//GVL.Drive1Settings[38].value:=80250;
//GVL.Drive1Settings[39].setting:='ACCE';
//GVL.Drive1Settings[39].value:=65535;
//GVL.Drive1Settings[40].setting:='DECE';
//GVL.Drive1Settings[40].value:=10000;
//GVL.Drive1Settings[41].setting:='PATH';
//GVL.Drive1Settings[41].value:=1;
//GVL.Drive1Settings[42].setting:='SLIM';
//GVL.Drive1Settings[42].value:=100000;
//GVL.Drive1Settings[43].setting:='ACTD';
//GVL.Drive1Settings[43].value:=1;


// Drive 2
GVL.Drive2Settings[0].setting:='4PHS';
GVL.Drive2Settings[0].value:=0;
//GVL.Drive2Settings[1].setting:='LLIM';
//GVL.Drive2Settings[1].value:=-40000;
//GVL.Drive2Settings[2].setting:='HLIM';
//GVL.Drive2Settings[2].value:=40001;
//GVL.Drive2Settings[3].setting:='ENCD';
//GVL.Drive2Settings[3].value:=1;
//GVL.Drive2Settings[4].setting:='ENCO';
//GVL.Drive2Settings[4].value:=0;
//GVL.Drive2Settings[5].setting:='INDA';
//GVL.Drive2Settings[5].value:=0;
//GVL.Drive2Settings[6].setting:='ISPD';
//GVL.Drive2Settings[6].value:=15000;
//GVL.Drive2Settings[7].setting:='ILIM';
//GVL.Drive2Settings[7].value:=3000;
//GVL.Drive2Settings[8].setting:='FILE';
//GVL.Drive2Settings[8].value:=0;
//GVL.Drive2Settings[9].setting:='ZON1';
//GVL.Drive2Settings[9].value:=100;
//GVL.Drive2Settings[10].setting:='ZON2';
//GVL.Drive2Settings[10].value:=1000;
//delta_zone := GVL.Drive2Settings[10].value - GVL.Drive2Settings[9].value;
//GVL.Drive2Settings[11].setting:='FREQ';
//GVL.Drive2Settings[11].value:=87000;
//GVL.Drive2Settings[12].setting:='FRQ2';
//GVL.Drive2Settings[12].value:=86000;
//GVL.Drive2Settings[13].setting:='FRAT';
//IF delta_zone = 0 THEN
//	GVL.Drive2Settings[13].value:=0;
//ELSE
//	GVL.Drive2Settings[13].value:= 65536 * (GVL.Drive2Settings[11].value - GVL.Drive2Settings[12].value) / delta_zone;	//145635;
//END_IF
//GVL.Drive2Settings[14].setting:='PROP';
//GVL.Drive2Settings[14].value:=20;
//GVL.Drive2Settings[15].setting:='PRO2';
//GVL.Drive2Settings[15].value:=10;
//GVL.Drive2Settings[16].setting:='PRAT';
//IF delta_zone = 0 THEN
//	GVL.Drive2Settings[16].value:=0;
//ELSE
//	GVL.Drive2Settings[16].value:= 65536 * (GVL.Drive2Settings[14].value - GVL.Drive2Settings[15].value) / delta_zone;	//2184;
//END_IF
//GVL.Drive2Settings[17].setting:='INTF';
//GVL.Drive2Settings[17].value:=15;
//GVL.Drive2Settings[18].setting:='CFRQ';
//GVL.Drive2Settings[18].value:=30000; //30000
//GVL.Drive2Settings[19].setting:='DUCO';
//GVL.Drive2Settings[19].value:=1;
//GVL.Drive2Settings[20].setting:='PTOL';
//GVL.Drive2Settings[20].value:=160;
//GVL.Drive2Settings[21].setting:='PTO2';
//GVL.Drive2Settings[21].value:=160;
//GVL.Drive2Settings[22].setting:='PHAC';
//GVL.Drive2Settings[22].value:=0;
//GVL.Drive2Settings[23].setting:='MIMP';
//GVL.Drive2Settings[23].value:=5000;
//GVL.Drive2Settings[24].setting:='MAMP';
//GVL.Drive2Settings[24].value:=65535;
//GVL.Drive2Settings[25].setting:='SLOP';
//GVL.Drive2Settings[25].value:= (GVL.Drive2Settings[24].value - GVL.Drive2Settings[23].value) / 192; //312;
//GVL.Drive2Settings[26].setting:='SOFS';
//GVL.Drive2Settings[26].value:= GVL.Drive2Settings[23].value - 64 * GVL.Drive2Settings[25].value; //-14968;
//GVL.Drive2Settings[27].setting:='FILA';
//GVL.Drive2Settings[27].value:=1;
//GVL.Drive2Settings[28].setting:='FILP';
//GVL.Drive2Settings[28].value:=1;
//GVL.Drive2Settings[29].setting:='AMPL';
//GVL.Drive2Settings[29].value:=65535;
//GVL.Drive2Settings[30].setting:='PHAS';
//GVL.Drive2Settings[30].value:=16383;
//GVL.Drive2Settings[31].setting:='TOUT';
//GVL.Drive2Settings[31].value:=500;
//GVL.Drive2Settings[32].setting:='TOU2';
//GVL.Drive2Settings[32].value:=0;
//GVL.Drive2Settings[33].setting:='TOU3';
//GVL.Drive2Settings[33].value:=7000;
//GVL.Drive2Settings[34].setting:='ELIM';
//GVL.Drive2Settings[34].value:=0;
//GVL.Drive2Settings[35].setting:='BLCK';
//GVL.Drive2Settings[35].value:=0;
//GVL.Drive2Settings[36].setting:='DLAY';
//GVL.Drive2Settings[36].value:=5;
//GVL.Drive2Settings[37].setting:='DTIM';
//GVL.Drive2Settings[37].value:=0;
//GVL.Drive2Settings[38].setting:='SSPD';
//GVL.Drive2Settings[38].value:=150000;
//GVL.Drive2Settings[39].setting:='ACCE';
//GVL.Drive2Settings[39].value:=10000;
//GVL.Drive2Settings[40].setting:='DECE';
//GVL.Drive2Settings[40].value:=10000;
//GVL.Drive2Settings[41].setting:='PATH';
//GVL.Drive2Settings[41].value:=0;
//GVL.Drive2Settings[42].setting:='SLIM';
//GVL.Drive2Settings[42].value:=100000;
//GVL.Drive2Settings[43].setting:='ACTD';
//GVL.Drive2Settings[43].value:=0;

GVL.Drive3Settings[0].setting:='4PHS';
GVL.Drive3Settings[0].value:=0;

GVL.Drive4Settings[0].setting:='4PHS';
GVL.Drive4Settings[0].value:=0;
END_IF

END_PROGRAM

// ---- GlobalTextList.TcGTLO
TEXTLIST GlobalTextList
  740 = "\n{attribute 'to_string'}"
  145 = '%s'
  522 = '-'
  680 = '4'
  265 = 'Acc'
  284 = 'Act'
  645 = 'Actual position'
  651 = 'Amp En'
  9 = 'Dec'
  357 = 'DEMO'
  240 = 'DIR'
  529 = 'Done'
  918 = 'DPOS'
  323 = 'DRIVE 1'
  129 = 'Drive 1'
  156 = 'DRIVE 2'
  599 = 'Drive 2'
  338 = 'DRIVE 3'
  828 = 'DRIVE 4'
  710 = 'ENABLE'
  360 = 'Enabled'
  608 = 'ENBL'
  426 = 'ENCR'
  659 = 'End stop'
  6 = 'End stop L'
  818 = 'End stop left'
  937 = 'End stop R'
  802 = 'End stop Right'
  649 = 'End stop right'
  465 = 'Error'
  633 = 'etTarg'
  435 = 'HALSTOP'
  447 = 'HALT'
  688 = 'Has iIndex'
  609 = 'Has Index'
  73 = 'Has index'
  610 = 'Index'
  553 = 'INDEX'
  505 = 'Indexdex'
  920 = 'INDX'
  717 = 'INIT'
  864 = 'JOG'
  548 = 'JOG+'
  123 = 'JOG-'
  124 = 'Left end stop'
  925 = 'Motor  On'
  113 = 'Motor End stop'
  817 = 'Motor On'
  344 = 'MOVE '
  578 = 'MOVE +'
  436 = 'MOVE+'
  355 = 'MOVE-'
  580 = 'Pos ReachDone'
  577 = 'Pos Reached'
  786 = 'RESET'
  567 = 'RST'
  752 = 'SCAN'
  449 = 'Speed'
  524 = 'STOP'
  343 = 'Targ'
  711 = 'Target'
END_TEXTLIST

// ---- VISUs/Visualization.TcVIS
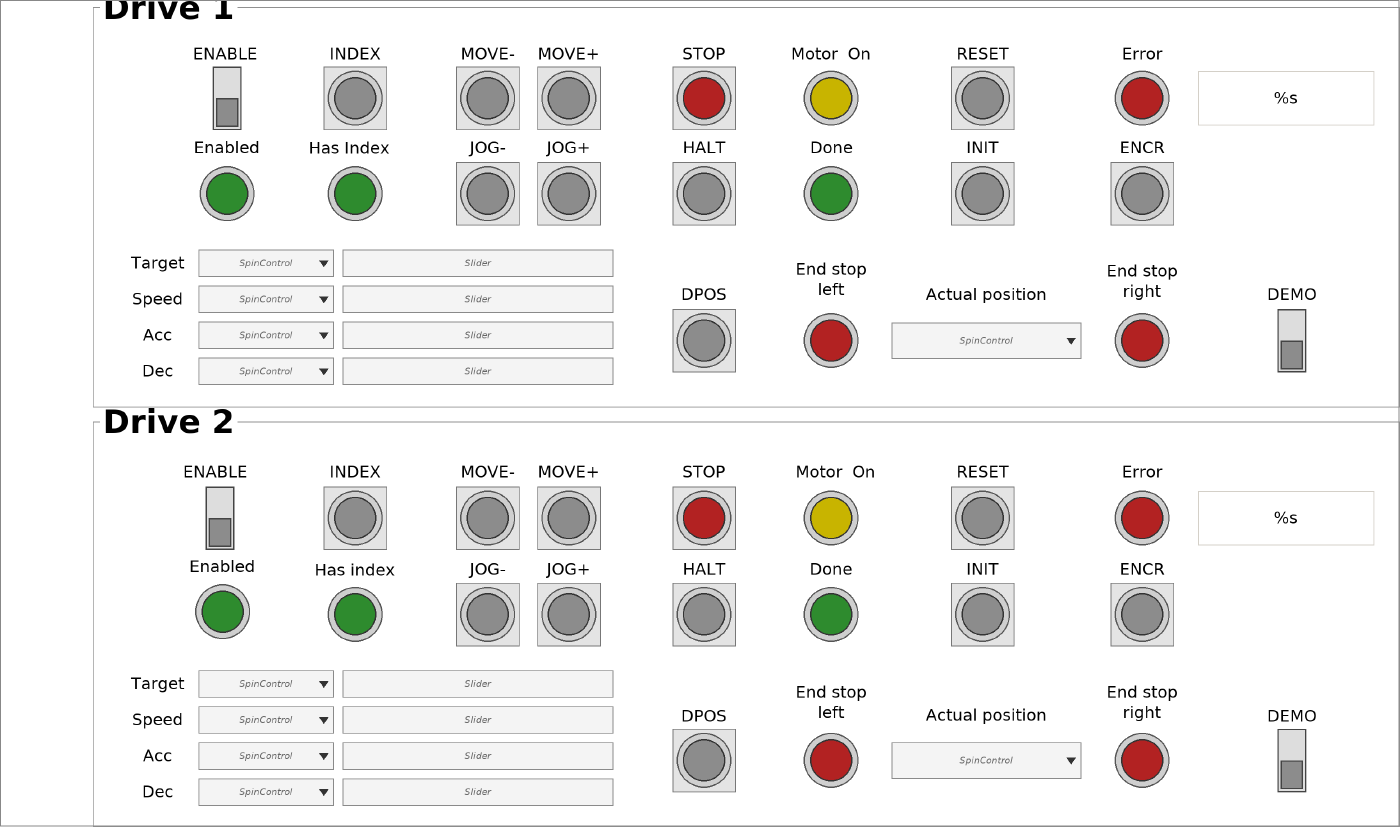
VISUALIZATION Visualization  // 1553x918
    GroupBox (103,0 1450x452), "Drive 1"
        Label (222,136 125x57), "Has Index"
        Label (762,33 114x54), "Motor On"
        PushSwitch (643,343 70x70), variable: MAIN.drive1Dpos, behaviour: TAP, style: Switch-PushSwitch-Gray
        Label (643,312 70x30), "DPOS"
        Textfield (1226,79 195x60), "%s", text variable: MAIN.drive1ErrorString
    GroupBox (103,460 1450x458), "Drive 2"
        Label (232,145 117x56), "Has index"
        Lamp1 (109,184 70x70), variable: MAIN.Drive2.iDriveAmplifiersEnabled, style: Lamp-Lamp1-Green
        Label (92,154 103x30), "Enabled"
        Label (769,38 110x52), "Motor On"
        PushSwitch (643,349 70x70), variable: MAIN.drive2Dpos, behaviour: TAP, style: Switch-PushSwitch-Gray
        Label (643,320 70x30), "DPOS"
        Label (907,319 168x30), "Actual position"
        Textfield (1226,85 195x60), "%s", text variable: MAIN.drive2ErrorString
    DipSwitch (1398,343 70x70), variable: MAIN.drive1MoveAbs, behaviour: TOGGLE, style: Switch-DipSwitch-Gray
    SpinControl (220,317 150x30), variable: MAIN.drive1Speed
    SpinControl (220,357 150x30), variable: MAIN.drive1Acc
    SpinControl (220,277 150x30), variable: MAIN.drive1Target
    SpinControl (220,397 150x30), variable: MAIN.drive1Dec
    Lamp1 (887,74 70x70), variable: MAIN.Drive1.MotorOn, style: Lamp-Lamp1-Yellow
    Lamp1 (1232,343 70x70), variable: MAIN.Drive1.RightEndstop, style: Lamp-Lamp1-Red
    Lamp1 (887,343 70x70), variable: MAIN.Drive1.LeftEndstop, style: Lamp-Lamp1-Red
    PushSwitch (1055,74 70x70), variable: MAIN.drive1Reset, behaviour: TAP, style: Switch-PushSwitch-Gray
    PushSwitch (746,74 70x70), variable: MAIN.drive1Stop, behaviour: TAP, style: Switch-PushSwitch-Red
    PushSwitch (746,180 70x70), variable: MAIN.drive1Halt, behaviour: TAP, style: Switch-PushSwitch-Gray
    PushSwitch (359,74 70x70), variable: MAIN.drive1Index, behaviour: TAP, style: Switch-PushSwitch-Gray
    Label (1388,312 90x30), "DEMO"
    Label (359,45 70x30), "INDEX"
    Label (746,149 70x30), "HALT"
    Label (746,45 70x30), "STOP"
    Label (1055,45 70x30), "RESET"
    Lamp1 (887,180 70x70), variable: MAIN.Drive1.Done, style: Lamp-Lamp1-Green
    Label (872,278 100x64), "End stop left"
    Label (1217,282 100x60), "End stop right"
    Label (877,149 91x30), "Done"
    Label (140,277 70x30), "Target"
    Label (140,317 70x30), "Speed"
    Label (140,357 70x30), "Acc"
    Label (140,397 70x30), "Dec"
    Label (1013,312 162x30), "Actual position"
    SpinControl (989,358 210x40), variable: MAIN.Drive1.ActPosition
    Slider (380,277 300x30), variable: MAIN.drive1Target, scale 0..100
    Slider (380,317 300x30), variable: MAIN.drive1Speed, scale 0..100
    Slider (380,357 300x30), variable: MAIN.drive1Acc, scale 0..100
    Slider (380,397 300x30), variable: MAIN.drive1Dec, scale 0..100
    DipSwitch (1398,809 70x70), variable: MAIN.drive2MoveAbs, behaviour: TOGGLE, style: Switch-DipSwitch-Gray
    SpinControl (220,784 150x30), variable: MAIN.drive2Speed
    SpinControl (220,824 150x30), variable: MAIN.drive2Acc
    SpinControl (220,744 150x30), variable: MAIN.drive2Target
    SpinControl (220,864 150x30), variable: MAIN.drive2Dec
    Lamp1 (887,540 70x70), variable: MAIN.Drive2.MotorOn, style: Lamp-Lamp1-Yellow
    Lamp1 (1232,809 70x70), variable: MAIN.Drive2.RightEndstop, style: Lamp-Lamp1-Red
    Lamp1 (887,809 70x70), variable: MAIN.Drive2.LeftEndstop, style: Lamp-Lamp1-Red
    PushSwitch (1055,540 70x70), variable: MAIN.drive2Reset, behaviour: TAP, style: Switch-PushSwitch-Gray
    PushSwitch (746,540 70x70), variable: MAIN.drive2Stop, behaviour: TAP, style: Switch-PushSwitch-Red
    PushSwitch (746,647 70x70), variable: MAIN.drive2Halt, behaviour: TAP, style: Switch-PushSwitch-Gray
    PushSwitch (359,540 70x70), variable: MAIN.drive2Index, behaviour: TAP, style: Switch-PushSwitch-Gray
    Label (1388,780 90x30), "DEMO"
    Label (359,509 70x30), "INDEX"
    Label (746,617 70x30), "HALT"
    Label (746,509 70x30), "STOP"
    Label (1055,509 70x30), "RESET"
    Lamp1 (887,647 70x70), variable: MAIN.Drive2.Done, style: Lamp-Lamp1-Green
    Label (872,749 100x61), "End stop left"
    Label (1217,749 100x61), "End stop right"
    Label (875,617 94x30), "Done"
    Label (140,744 70x30), "Target"
    Label (140,784 70x30), "Speed"
    Label (140,824 70x30), "Acc"
    Label (140,864 70x30), "Dec"
    SpinControl (989,824 210x40), variable: MAIN.Drive2.ActPosition
    Slider (380,744 300x30), variable: MAIN.drive2Target, scale 0..100
    Slider (380,784 300x30), variable: MAIN.drive2Speed, scale 0..100
    Slider (380,824 300x30), variable: MAIN.drive2Acc, scale 0..100
    Slider (380,864 300x30), variable: MAIN.drive2Dec, scale 0..100
    DipSwitch (217,74 70x70), variable: MAIN.drive1Enable, behaviour: TOGGLE, style: Switch-DipSwitch-Gray
    Label (200,45 100x30), "ENABLE"
    Label (189,509 100x30), "ENABLE"
    DipSwitch (209,540 70x70), variable: MAIN.drive2Enable, behaviour: TOGGLE, style: Switch-DipSwitch-Gray
    Lamp1 (359,180 70x70), variable: MAIN.Drive1.HasIndex, style: Lamp-Lamp1-Green
    Lamp1 (359,647 70x70), variable: MAIN.Drive2.HasIndex, style: Lamp-Lamp1-Green
    PushSwitch (506,180 70x70), variable: MAIN.drive1JogN, behaviour: TAP, style: Switch-PushSwitch-Gray
    PushSwitch (596,180 70x70), variable: MAIN.drive1JogP, behaviour: TAP, style: Switch-PushSwitch-Gray
    Label (506,149 70x30), "JOG-"
    Label (596,149 70x30), "JOG+"
    PushSwitch (506,647 70x70), variable: MAIN.drive2JogN, behaviour: TAP, style: Switch-PushSwitch-Gray
    PushSwitch (596,647 70x70), variable: MAIN.drive2JogP, behaviour: TAP, style: Switch-PushSwitch-Gray
    Label (506,617 70x30), "JOG-"
    Label (596,617 70x30), "JOG+"
    PushSwitch (1055,180 70x70), variable: MAIN.drive1Init, behaviour: TAP, style: Switch-PushSwitch-Gray
    Label (1055,149 70x30), "INIT"
    PushSwitch (1055,647 70x70), variable: MAIN.drive2Init, behaviour: TAP, style: Switch-PushSwitch-Gray
    Label (1055,617 70x30), "INIT"
    Lamp1 (1232,74 70x70), variable: MAIN.Drive1.HasError, style: Lamp-Lamp1-Red
    Label (1217,45 100x30), "Error"
    Lamp1 (1232,540 70x70), variable: MAIN.Drive2.HasError, style: Lamp-Lamp1-Red
    Label (1217,509 100x30), "Error"
    Lamp1 (217,180 70x70), variable: MAIN.Drive1.iDriveAmplifiersEnabled, style: Lamp-Lamp1-Green
    Label (200,149 103x30), "Enabled"
    PushSwitch (506,74 70x70), variable: MAIN.drive1MoveN, behaviour: TAP, style: Switch-PushSwitch-Gray
    PushSwitch (596,74 70x70), variable: MAIN.drive1MoveP, behaviour: TAP, style: Switch-PushSwitch-Gray
    Label (506,45 70x30), "MOVE-"
    Label (596,45 70x30), "MOVE+"
    PushSwitch (1232,180 70x70), variable: MAIN.drive1ResetEncoder, behaviour: TAP, style: Switch-PushSwitch-Gray
    Label (1223,149 88x30), "ENCR"
    PushSwitch (1232,647 70x70), variable: MAIN.drive2ResetEncoder, behaviour: TAP, style: Switch-PushSwitch-Gray
    Label (1223,617 88x30), "ENCR"
    PushSwitch (506,540 70x70), variable: MAIN.drive2MoveN, behaviour: TAP, style: Switch-PushSwitch-Gray
    PushSwitch (596,540 70x70), variable: MAIN.drive2MoveP, behaviour: TAP, style: Switch-PushSwitch-Gray
    Label (506,509 70x30), "MOVE-"
    Label (596,509 70x30), "MOVE+"
END_VISUALIZATION
